Staubli VAL3: Entwicklungsmethodik.dtx

mdesc mNomSpeed
frame fUserFrame = {x=1007.262395, y=-312.843264, z=-186.866453, rx=-0.535332, ry=-0.21904, rz=90.124968, fatherId=world[0]}
sio soTcpClient = {link=Socket\server0}
jointRx jHome = {j3=90, j5=90}
bool bNewData
num nData[5]
bool bReady
tool tGreiferM = {y=-27, z=127, rx=45, fatherId=flange[0], ioLink=ValveIO\valve1, ioOpen=0.05, ioClose=0.05}
tool tGreiferS = {y=27, z=127, rx=-45, ry=5.50371872946114E-07, rz=179.999999432294, fatherId=flange[0], ioLink=ValveIO\valve1, ioOpen=0.05, ioClose=0.05}
bool bVereinzeln
bool bPick
trsf trApro = {z=-150}
pointRx pPick[4]
  [0] = {z=6, rx=180, rz=45, fatherId=fUserFrame[0]}
  [1] = {z=20, rx=180, rz=45, fatherId=fUserFrame[0]}
  [2] = {z=6, rx=180, rz=45, fatherId=fUserFrame[0]}
  [3] = {z=10, rx=180, rz=45, fatherId=fUserFrame[0]}
mdesc mUsedSpeed
pointRx pPlace = {z=50, rx=180, rz=45, fatherId=fUserFrame[0]}
num nObj
num nOrientation
num nX
num nY
num nAngle
pointRx pVereinzeln = {z=10, rx=180, rz=45, fatherId=fUserFrame[0]}
trsf trVer = {x=100}
mdesc mVereinzeln = {accel=10, leave=1, reach=1}
num nX_S
num nX_M
num nY_M
num nY_S
dio delta_Y
dio delta_X
pointRx pEmpty = {fatherId=fUserFrame[0]}
jointRx jEmpty
pointRx pObj[10]
  [0] = {x=345, y=445, rz=350, fatherId=fUserFrame[0]}
  [1] = {x=256, y=423, rz=348, fatherId=fUserFrame[0]}
  [2] = {x=144, y=415, rz=354, fatherId=fUserFrame[0]}
  [3] = {x=71, y=410, rz=323, fatherId=fUserFrame[0]}
  [4] = {x=449, y=370, rz=224, fatherId=fUserFrame[0]}
  [5] = {x=163, y=356, rz=335, fatherId=fUserFrame[0]}
  [6] = {x=347, y=337, rz=182, fatherId=fUserFrame[0]}
  [7] = {x=84, y=333, rz=333, fatherId=fUserFrame[0]}
  [8] = {x=263, y=246, rz=523, fatherId=fUserFrame[0]}
  [9] = {x=406, y=235, rz=511, fatherId=fUserFrame[0]}
pointRx pAblegen[2]
  [0] = {x=700, y=125, fatherId=fUserFrame[0]}
  [1] = {x=700, y=375, fatherId=fUserFrame[0]}
